(* PLC project Simulation.project, CODESYS CODESYS V3.5 SP19 Patch 5 *)
(* stored: creationDateTime 2024-05-15T19:26:43.8609959, modificationDateTime 2023-08-21T12:28:56 *)

PROGRAM PLC_PRG
  VAR
    S1 : BOOL;
    S2 : BOOL;
    L1 : BOOL;
  END_VAR

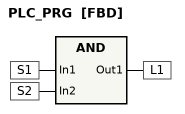
(* FBD diagram, written out as Structured Text *)
L1 := S1 AND S2;
END_PROGRAM

CONFIGURATION Device
  RESOURCE Application ON PLC
    TASK MainTask(INTERVAL := T#20ms, PRIORITY := 1);
    PROGRAM PLC_PRG WITH MainTask : PLC_PRG;
  END_RESOURCE
END_CONFIGURATION
